FUNCTION_BLOCK NullCoeDevice EXTENDS CyclicComponent IMPLEMENTS I_CoeDevice
VAR
END_VAR

PROPERTY AdsAddr : REFERENCE TO AMSADDR
GET
END_GET
SET
END_SET
END_PROPERTY

{attribute 'monitoring' := 'call'}
PROPERTY Busy : BOOL
GET
END_GET
END_PROPERTY

METHOD CyclicLogic
END_METHOD

{attribute 'monitoring' := 'call'}
PROPERTY Error : BOOL
GET
END_GET
END_PROPERTY

{attribute 'monitoring' := 'call'}
PROPERTY ErrorId : UDINT
GET
END_GET
END_PROPERTY

METHOD Read
VAR_INPUT
	Index	 : WORD;
	SubIndex : BYTE;
	pDstBuf	 : PVOID;
	BufLen	 : UDINT;
END_VAR
END_METHOD

METHOD Write
VAR_INPUT
	Index	 : WORD;
	SubIndex : BYTE;
	pDstBuf	 : PVOID;
	BufLen	 : UDINT;
END_VAR
END_METHOD

END_FUNCTION_BLOCK

(* stored: Version 1.1.0.1, ProductVersion 3.1.4026.18
   POU NullCoeDevice: Id {cc51e621-3816-4ad7-9cb7-05ab19309e13}, SpecialFunc None
   Property AdsAddr: Id {ceaec292-550a-4193-a150-cd2c4f832603}
   Get Get: Id {c2a6b1c7-30a3-4fa1-ba85-66af66662f12}
   Set Set: Id {963be93b-3880-4750-9cb6-559d2e63c047}
   Property Busy: Id {f1b6a8a3-071d-4baa-a1f9-a072e8db17b0}
   Get Get: Id {a7953960-2a08-4346-9ab7-415cb2392be5}
   Method CyclicLogic: Id {bb2b467e-e8db-4aa6-ab4e-f0c8e4749e79}
   Property Error: Id {0ec2ecc3-3e82-469a-8366-e49550b7ca40}
   Get Get: Id {6339ce2b-154e-40da-823f-06898841d16d}
   Property ErrorId: Id {dea5f65f-b3ed-4838-b89c-05989f95cf9e}
   Get Get: Id {2d022af6-c5c6-48e6-b473-7be263f3ec03}
   Method Read: Id {ff6fa20a-815f-4927-bc2c-5640028c35e0}
   Method Write: Id {e0d6c901-56a2-4d7f-b7d9-b39556a02436} *)
